INTERFACE I_DictionaryTreeNode EXTENDS I_CollectionNode

METHOD PUBLIC Clone
VAR_INPUT
	Node : I_DictionaryTreeNode;
END_VAR
END_METHOD

PROPERTY PUBLIC Height : DINT
GET
END_GET
SET
END_SET
END_PROPERTY

METHOD Initialize
VAR_INPUT
	Key : T_MAXSTRING;
	Value : ANY;
END_VAR
END_METHOD

PROPERTY PUBLIC Key : T_MAXSTRING
GET
END_GET
END_PROPERTY

PROPERTY PUBLIC Left : I_DictionaryTreeNode
GET
END_GET
SET
END_SET
END_PROPERTY

PROPERTY PUBLIC NodeBufferPointer : Pointer To Byte
GET
END_GET
END_PROPERTY

PROPERTY PUBLIC NodeBufferSize : UDINT
GET
END_GET
END_PROPERTY

PROPERTY PUBLIC Right : I_DictionaryTreeNode
GET
END_GET
SET
END_SET
END_PROPERTY

END_INTERFACE

(* stored: Version 1.1.0.1, ProductVersion 3.1.4024.12
   Itf I_DictionaryTreeNode: Id {b049ebc5-6910-459d-8181-35c0e92ce9cc}
   Method Clone: Id {5fbd90f7-ad8c-4844-a236-694402648117}
   Property Height: Id {d505bf5b-8ee9-455b-961d-2af3f83e2374}
   Get Get: Id {82350a15-c594-4ff4-89f1-edf1aa8dd241}
   Set Set: Id {5b56c20a-56a2-4da9-b79a-d9ab2cc0f075}
   Method Initialize: Id {4e666a69-fbdc-4504-8413-4d645bb072e7}
   Property Key: Id {346641d0-7fb0-4dfa-81c9-7410426c1415}
   Get Get: Id {2fa95320-2e04-46a8-9ef1-8c5876f59e56}
   Property Left: Id {a06887f7-f336-4b50-bf5c-920e26d04b52}
   Get Get: Id {290a01ba-12a0-4ac0-9463-c22efd8de14b}
   Set Set: Id {64bd001e-c04a-4304-9bf2-7a10ee37d04f}
   Property NodeBufferPointer: Id {d117737e-cc0e-4e5e-8a0b-d67defb04ced}
   Get Get: Id {92f300c7-46ed-421b-98d6-4b1eb2c5a56f}
   Property NodeBufferSize: Id {b53a213b-7a12-401e-bd14-fcbbc65ec2b1}
   Get Get: Id {fd927efb-202c-4042-8bd4-77eae35c8d58}
   Property Right: Id {4785ac1a-33ef-4008-9184-6e0b82817986}
   Get Get: Id {8d25d25a-0ad1-4409-ba9c-7468ae0f0930}
   Set Set: Id {0f893abf-81b1-4c64-a0b7-52ceb220507c} *)
